Staubli VAL3: sortObjects.pgx

program sortObjects(num x_nNumOfPart)
  local num l_nI
  local num l_nMaxIndex
  local num l_nJ
  local num l_nMaxValue
begin
  // This program sorts the parts from the part with the largest X
  //  value to the smallest X value. This particular order is
  //  convenient when the orientation of the detection frame has the
  //  same orientation as the conveyor frame because the first part
  //  on the queue should be the first part to arrive into the
  //  tracking window.
  //
  //----------------------------------------------------------------
  //
  // Init variables
  l_nMaxIndex=0
  //
  // Sort parts from the largest X to the smallest X
  for l_nJ=0 to x_nNumOfPart-1
    // Find the largest X
    l_nMaxValue=-power(2,100)
    for l_nI=0 to x_nNumOfPart-1
      if trObjectPos[l_nI].x>l_nMaxValue and nObjectID[l_nI]>0
        l_nMaxValue=trObjectPos[l_nI].x
        l_nMaxIndex=l_nI
      endIf
    endFor
    // Copy largest
    oTempQueue[l_nJ].nID=nObjectID[l_nMaxIndex]
    oTempQueue[l_nJ].trTrsf=trObjectPos[l_nMaxIndex]
    oTempQueue[l_nJ].nLatchedValue=nLatchedValue[l_nMaxIndex]
    // Erase largest
    nObjectID[l_nMaxIndex]=-1
  endFor
  //
  // Copy sorted values
  for l_nI=0 to x_nNumOfPart-1
    nObjectID[l_nI]=oTempQueue[l_nI].nID
    trObjectPos[l_nI]=oTempQueue[l_nI].trTrsf
    nLatchedValue[l_nI]=oTempQueue[l_nI].nLatchedValue
  endFor
end
